Staubli VAL3: chkDrvState.pgx

program chkDrvState(num x_nAxisNum)
  local num l_nStatus
  local num l_nStatus1
  local bool l_bIsOneBitSet
begin
  //检查状态
  l_nStatus=0
  //确定电机是否在remote状态
  // read status_remote register
  //  call chkStatusRemote(x_nAxisNum,l_bIsOneBitSet)
  //  if l_bIsOneBitSet
  //    nDrvState[x_nAxisNum]=15
  //  else

  //读取状态字
  call chkStatusWord(x_nAxisNum,l_nStatus)
  //cst:nDRV_ACTIV:掩码，111dec=1101111bin.驱动器处于某种状态
  l_nStatus1=bAnd(l_nStatus,cst:nDRV_ACTIV)
  switch l_nStatus1
    //
    case cst:nRdy2SwitchON
      nDrvState[x_nAxisNum]=3
    break
    //
    case cst:nSwitchedON
      nDrvState[x_nAxisNum]=4
    break
    //使能
    case cst:nOperatEnabled
      nDrvState[x_nAxisNum]=5
    break
    //quickstop
    case cst:nQuickStopActiv
      nDrvState[x_nAxisNum]=12
    break
    //
    default
      //cst:nDRV_FAULT=100 1111
      l_nStatus1=bAnd(l_nStatus,cst:nDRV_FAULT)

      switch l_nStatus1
        case cst:nNotRdySwiON
          nDrvState[x_nAxisNum]=1
        break
        //
        case cst:nSwitchONDis
          nDrvState[x_nAxisNum]=2
        break
        //
        case cst:nFaultReacActiv
          nDrvState[x_nAxisNum]=13
        break
        //
        case cst:nFaultState
          nDrvState[x_nAxisNum]=14
        break
        //
        default
          nDrvState[x_nAxisNum]=-1
        break
      endSwitch
    break
    //
  endSwitch
end
